{attribute 'qualified_only'}
{attribute 'strict'}
TYPE EFeedbackMsgAttenuationELL9 :
(
	StateMsg := 1,
	StatusMsg := 2,
	IsAliveMsg := 3,
	PositionMsg := 10,	
    IdMsg,
    CustomMsg	
);
END_TYPE

(* stored: Version 1.1.0.1, ProductVersion 3.1.4024.12
   DUT EFeedbackMsgAttenuationELL9: Id {14b5d664-2a58-4ab2-8e0e-86609c2cf279} *)
